{attribute addProperty BoxType "EK1122-0000-0018"}
{attribute addProperty Id "Beckhoff_EK13xxsub_EK1100EK1100_179A0949162A_0001_EK1300_0000_0017EK1300_0EEAC8F2344.25"}
{attribute addProperty CRC "2021904768"}
{attribute addProperty SizeInBites "50"}
{attribute addProperty SizeInBytes "6.25"}
TYPE Beckhoff_EK13xxEK1122_7883D180 EXTENDS EK1122_179A0949 :
STRUCT
	{attribute addProperty Name "Beckhoff_EK13xxsub_EK1100"}
	Beckhoff_EK13xxsub_EK1100 : EK1100_179A0949;
	{attribute addProperty Name "A_0001_EK1300_0000_0017"}
	A_0001_EK1300_0000_0017 : EK1300_0EEAC8F2;
END_STRUCT
END_TYPE

(* stored: Version 1.2.0.0, ProductVersion 3.1.4024.9
   DUT Beckhoff_EK13xxEK1122_7883D180: Id {58d44196-c191-4d21-bddb-99fec3a88fcd} *)
